(* IEC 61131-3 sources: JaccoSigma/tempclass/Class/VST011 (part 2) *)

      //LowLomit
      if FrequencyLimit8 > FrequencyBandwidth / 2 then
        a_FrequencyLimit[3].LimitLow := FrequencyLimit8 - (FrequencyBandwidth / 2);
      else
        a_FrequencyLimit[3].LimitLow := FrequencyLimit8;
      end_if;

      //High Limit
      if FrequencyLimit8 + (FrequencyBandwidth / 2) < 1000000 then
        a_FrequencyLimit[3].LimitHigh  := FrequencyLimit8 + (FrequencyBandwidth / 2);
      else
        a_FrequencyLimit[3].LimitHigh := FrequencyLimit8;
      end_if;

    else

      //Set inactive
      a_FrequencyLimit[3].LimitHigh := a_FrequencyLimit[3].LimitLow := 16#FFFF_FFFF;

    end_if;

  end_if;

  result := input;

END_FUNCTION

FUNCTION VIRTUAL GLOBAL VST011::FrequencyLimit16::Write
  VAR_INPUT
    input (EAX)   : UDINT;
  END_VAR
  VAR_OUTPUT
    result (EAX)  : UDINT;
  END_VAR

  // Max Frequency is 1 Mhz
  IF input > 1000000 & input <> 16#FFFF_FFFF THEN
    input := 1000000;
  END_IF;

  if FrequencyLimit16 <> input then //do we have a new value?

    //Save Input
    FrequencyLimit16 := input;

    //Set new Limit
    WriteParameter(us_ParameterNr:= VST_ASYNC_FREQUENCYLIMIT16, ud_Value:=FrequencyLimit16);

    //Calculate Limits for Hysterese
    //*****************************************************************************
    if FrequencyLimit16 <> 16#FFFF_FFFF then

      //LowLomit
      if FrequencyLimit16 > FrequencyBandwidth / 2 then
        a_FrequencyLimit[4].LimitLow := FrequencyLimit16 - (FrequencyBandwidth / 2);
      else
        a_FrequencyLimit[4].LimitLow := FrequencyLimit16;
      end_if;

      //High Limit
      if FrequencyLimit16 + (FrequencyBandwidth / 2) < 1000000 then
        a_FrequencyLimit[4].LimitHigh  := FrequencyLimit16 + (FrequencyBandwidth / 2);
      else
        a_FrequencyLimit[4].LimitHigh := FrequencyLimit16;
      end_if;

    else

      //Set inactive
      a_FrequencyLimit[4].LimitHigh := a_FrequencyLimit[4].LimitLow := 16#FFFF_FFFF;

    end_if;

  end_if;

  result := input;

END_FUNCTION

FUNCTION VIRTUAL GLOBAL VST011::FrequencyLimit32::Write
  VAR_INPUT
    input (EAX)   : UDINT;
  END_VAR
  VAR_OUTPUT
    result (EAX)  : UDINT;
  END_VAR

  // Max Frequency is 1 Mhz
  IF input > 1000000 & input <> 16#FFFF_FFFF THEN
    input := 1000000;
  END_IF;

  if FrequencyLimit32 <> input then //do we have a new value?

    //Save Input
    FrequencyLimit32 := input;

    //Set new Limit
    WriteParameter(us_ParameterNr:= VST_ASYNC_FREQUENCYLIMIT32, ud_Value:=FrequencyLimit32);

    //Calculate Limits for Hysterese
    //*****************************************************************************
    if FrequencyLimit32 <> 16#FFFF_FFFF then

      //LowLomit
      if FrequencyLimit32 > FrequencyBandwidth / 2 then
        a_FrequencyLimit[5].LimitLow := FrequencyLimit32 - (FrequencyBandwidth / 2);
      else
        a_FrequencyLimit[5].LimitLow := FrequencyLimit32;
      end_if;

      //High Limit
      if FrequencyLimit32 + (FrequencyBandwidth / 2) < 1000000 then
        a_FrequencyLimit[5].LimitHigh  := FrequencyLimit32 + (FrequencyBandwidth / 2);
      else
        a_FrequencyLimit[5].LimitHigh := FrequencyLimit32;
      end_if;

    else

      //Set inactive
      a_FrequencyLimit[5].LimitHigh := a_FrequencyLimit[5].LimitLow := 16#FFFF_FFFF;

    end_if;

  end_if;

  result := input;

END_FUNCTION

FUNCTION VIRTUAL GLOBAL VST011::HWRampdownDeltaFrequency::Write
  VAR_INPUT
    input (EAX)   : DINT;
  END_VAR
  VAR_OUTPUT
    result (EAX)  : DINT;
  END_VAR

  WriteParameter(us_ParameterNr := VST_ASYNC_EXTERNALLOCKDELTAFREQUENCY, ud_Value := input$UDINT);
  result := input;

END_FUNCTION

FUNCTION VIRTUAL GLOBAL VST011::HWRampdownDeltaTime::Write
  VAR_INPUT
    input (EAX)   : DINT;
  END_VAR
  VAR_OUTPUT
    result (EAX)  : DINT;
  END_VAR

  WriteParameter(us_ParameterNr := VST_ASYNC_EXTERNALLOCKDELTATIME, ud_Value := input$UDINT);
  result := input;

END_FUNCTION

FUNCTION GLOBAL VST011::RequestParameter
  VAR_INPUT
    us_ParameterNr  : USINT;
  END_VAR
  VAR_OUTPUT
    retcode   : DINT;
  END_VAR
  VAR
    tmpCounter : USINT;
  END_VAR

  retcode := VST_ERROR_ASYNC_NOERROR;

  if us_ParameterNr <= VST011_MAXASYNCPARAMETER &  us_ReadNumber <= VST011_MAXASYNCPARAMETER then

    // Check if Element is already active
    //*****************************************************************************
    if us_ReadNumber then

      //No Overflow of Buffer (to be Thread-Safe)
      //---------------------------------------------------------------------------
      if us_ReadPosition + us_ReadNumber - 1 <= VST011_MAXASYNCPARAMETER then

        for tmpCounter := us_ReadPosition to us_ReadPosition + us_ReadNumber - 1 do
          if a_ParameterReadRequest[tmpCounter] = us_ParameterNr then
            retcode := VST_ERROR_ASYNC_ALREADYACTIVE;
            return;
          end_if;
        end_for;

      //Overflow of Buffer (to be Thread-Safe)
      //---------------------------------------------------------------------------
      else

        //Check actual Position to End of Buffer
        for tmpCounter := us_ReadPosition to VST011_MAXASYNCPARAMETER do
          if a_ParameterReadRequest[tmpCounter] = us_ParameterNr then
            retcode := VST_ERROR_ASYNC_ALREADYACTIVE;
            return;
          end_if;
        end_for;

        //Check from Zero to actual Element
        for tmpCounter := 0 to us_ReadNumber - VST011_MAXASYNCPARAMETER + us_ReadPosition - 2 do
          if a_ParameterReadRequest[tmpCounter] = us_ParameterNr then
            retcode := VST_ERROR_ASYNC_ALREADYACTIVE;
            return;
          end_if;
        end_for;
      end_if;

    end_if;

    // Save into Queue for asynchronous ReadAccess
    //*****************************************************************************
    if us_ReadPosition + us_ReadNumber <= VST011_MAXASYNCPARAMETER  then
      a_ParameterReadRequest[us_ReadPosition + us_ReadNumber]   := us_ParameterNr;
    else
      a_ParameterReadRequest[us_ReadPosition + us_ReadNumber - VST011_MAXASYNCPARAMETER - 1] := us_ParameterNr;
    end_if;

    us_ReadNumber += 1;
    a_ReadDataBuffer[us_ParameterNr].b_Valid := false;

  else
    retcode := VST_ERROR_ASYNC_INVALIDPARAMETER;
  end_if;

END_FUNCTION

FUNCTION GLOBAL VST011::WriteParameter
  VAR_INPUT
    us_ParameterNr  : USINT;
    ud_Value  : UDINT;
  END_VAR
  VAR_OUTPUT
    retcode   : DINT;
  END_VAR
  VAR
    tmpCounter : USINT;
    pAsyWrData  : ^t_AsyncWriteData;
    pLastWritten: ^t_LastWrittenValues;
    ForEnd : USINT;
  END_VAR

  retcode := VST_ERROR_ASYNC_NOERROR;

  IF (us_ParameterNr <= VST011_MAXASYNCPARAMETER) & (us_WriteNumber <= VST011_MAXASYNCPARAMETER) THEN
    CASE us_ParameterNr OF
      VST_ASYNC_INCREMENTALENCODERSETTINGS, //not implemented (user otherwise might access internal test-registers)
      VST_ASYNC_BRIDGE2OFF, //implemented but may not be called (user could damage the card)!
      VST_ASYNC_BRIDGE2MUL,
      VST_ASYNC_BRIDGE2DIV,
      VST_ASYNC_BRIDGE1OFF,
      VST_ASYNC_BRIDGE1MUL,
      VST_ASYNC_BRIDGE1DIV,
      VST_ASYNC_BRIDGESUPPLYVOLTAGELOWERTHRESHOLD,
      VST_ASYNC_BRIDGESUPPLYVOLTAGEUPPERTHRESHOLD,
      VST_ASYNC_BRIDGETEMPERATUREWARNINGTHRESHOLD,
      VST_ASYNC_BRIDGETEMPERATUREERRORTHRESHOLD,
      VST_ASYNC_EXTENDEDSTATEWORD,
      VST_ASYNC_COMMUTATIONCOUNTERBRIDGE1,
      VST_ASYNC_COMMUTATIONCOUNTERBRIDGE2,
      VST_ASYNC_ONTIMECOUNTERBRIDGE1,
      VST_ASYNC_ONTIMECOUNTERBRIDGE2,
      VST_ASYNC_HBRIDGE_VOLTAGE,
      VST_ASYNC_HBRIDGE_TEMPERATURE:
        retcode := VST_ERROR_ASYNC_WRITENOTALLOWED;
    ELSE
      // if the value is the same as the last value we wrote on this parameter => don't do it
      pLastWritten := #a_LastWrittenAsyValues[0] + us_ParameterNr * sizeof(t_LastWrittenValues);
      if (pLastWritten^.AlreadyUsed = TRUE) & (ud_Value = pLastWritten^.Value) then
        // this is already the actual value of this parameter
        return;
      end_if;

      // Check if Element is already active
      //*****************************************************************************
      if us_WriteNumber then

        //No Overflow of Buffer (to be Thread-Safe)
        //---------------------------------------------------------------------------
        if us_WritePosition + us_WriteNumber - 1 <= VST011_MAXASYNCPARAMETER then
          // calculate the end only once
          ForEnd := (us_WritePosition + us_WriteNumber - 1);
          pAsyWrData := #a_WriteDataBuffer[0] + us_WritePosition * sizeof(t_AsyncWriteData);
          for tmpCounter := us_WritePosition to ForEnd do
            if pAsyWrData^.us_ID = us_ParameterNr then
              retcode := VST_ERROR_ASYNC_ALREADYACTIVE;
              pAsyWrData^.ud_Value := ud_Value;
              return;
            end_if;
            pAsyWrData += sizeof(a_WriteDataBuffer);
          end_for;

        //Overflow of Buffer (to be Thread-Safe)
        //---------------------------------------------------------------------------
        else
          //Check actual Position to End of Buffer
          pAsyWrData := #a_WriteDataBuffer[0] + us_WritePosition * sizeof(t_AsyncWriteData);
          for tmpCounter := us_WritePosition to VST011_MAXASYNCPARAMETER do
            if pAsyWrData^.us_ID = us_ParameterNr then
              retcode := VST_ERROR_ASYNC_ALREADYACTIVE;
              pAsyWrData^.ud_Value := ud_Value;
              return;
            end_if;
            pAsyWrData += sizeof(t_AsyncWriteData);
          end_for;

          //Check from Zero to actual Element
          ForEnd := us_WriteNumber - VST011_MAXASYNCPARAMETER + us_WritePosition - 2;
          pAsyWrData := #a_WriteDataBuffer[0];
          for tmpCounter := 0 to ForEnd do
            if pAsyWrData^.us_ID = us_ParameterNr then
              retcode := VST_ERROR_ASYNC_ALREADYACTIVE;
              pAsyWrData^.ud_Value := ud_Value;
              return;
            end_if;
            pAsyWrData += sizeof(t_AsyncWriteData);
          end_for;
        end_if;

      end_if;

      // Save into Queue for asynchronous WriteAccess
      //*****************************************************************************
      if us_WritePosition + us_WriteNumber <= VST011_MAXASYNCPARAMETER  then
        pAsyWrData := #a_WriteDataBuffer[0] + (us_WritePosition + us_WriteNumber) * sizeof(t_AsyncWriteData);
      else
        pAsyWrData := #a_WriteDataBuffer[0] + (us_WriteNumber + us_WritePosition - VST011_MAXASYNCPARAMETER - 1) * sizeof(t_AsyncWriteData);
      end_if;

      pAsyWrData^.us_ID    := us_ParameterNr;
      pAsyWrData^.ud_Value := ud_Value;

      pLastWritten^.Value := ud_Value;
      pLastWritten^.AlreadyUsed := TRUE;

      us_WriteNumber += 1;
    END_CASE;
  ELSE
    retcode := VST_ERROR_ASYNC_INVALIDPARAMETER;
  END_IF;

END_FUNCTION

FUNCTION GLOBAL VST011::ReadParameter
  VAR_INPUT
    us_ParameterNr  : USINT;
    p_b_Valid   : ^BOOL;
    p_ud_Value  : ^UDINT;
  END_VAR
  VAR_OUTPUT
    retcode   : DINT;
  END_VAR

  retcode := VST_ERROR_ASYNC_NOERROR;

  IF us_ParameterNr <= VST011_MAXASYNCPARAMETER THEN
    IF p_b_Valid <> NIL THEN
      p_b_Valid^ := a_ReadDataBuffer[us_ParameterNr].b_Valid;
    END_IF;
    a_ReadDataBuffer[us_ParameterNr].b_Valid := FALSE;
    IF p_ud_Value <> NIL THEN
      p_ud_Value^ := a_ReadDataBuffer[us_ParameterNr].ud_Value;
    ELSE
      retcode := VST_ERROR_ASYNC_NOVALUEPTR;
    END_IF;
  ELSE
    retcode := VST_ERROR_ASYNC_INVALIDPARAMETER;
  END_IF;

END_FUNCTION

FUNCTION VIRTUAL GLOBAL VST011::MaxCurrent::Write
  VAR_INPUT
    input (EAX)   : DINT;
  END_VAR
  VAR_OUTPUT
    result (EAX)  : DINT;
  END_VAR

  //Check for Change
  if input <> MaxCurrent then

    //Check Limit
    if input < 0 then
      input := 0;
    elsif input > sd_MaxAllowedCurrent then
      input := sd_MaxAllowedCurrent;
    end_if;

    //Calculate Current
    if abs(SetFreqOut)$UDINT <= udStallCurrentWindow then
      u_MaxCurrent := to_uint(input - ((input * StallCurrentReduction) / 1000));
    else
      u_MaxCurrent := to_uint(input);
    end_if;

  end_if;

  result := MaxCurrent := input;

END_FUNCTION

FUNCTION VIRTUAL GLOBAL VST011::UpdateRetryCounter
  VAR
    tempRetryCounter : USINT;
  END_VAR

  // LanSte 16.04.2013 10:49
  // Updated to use new Method for Payload support
  tempRetryCounter := GetRetryCounter(ud_DOHandle := s_IODataObject.p_Handle$UDINT);
  if ( tempRetryCounter <> s_IODataObject.us_OldRetryCounter ) then
    RetryCounter += TO_USINT( tempRetryCounter - s_IODataObject.us_OldRetryCounter );
    s_IODataObject.us_OldRetryCounter := tempRetryCounter;
  end_if;

  tempRetryCounter := GetRetryCounter(ud_DOHandle := s_ISyncDO.p_Handle$UDINT);
  if ( tempRetryCounter <> s_ISyncDO.us_OldRetryCounter ) then
    RetryCounter += TO_USINT( tempRetryCounter - s_ISyncDO.us_OldRetryCounter );
    s_ISyncDO.us_OldRetryCounter := tempRetryCounter;
  end_if;

  tempRetryCounter := GetRetryCounter(ud_DOHandle := s_SettingsDataObject.p_Handle$UDINT);
  if ( tempRetryCounter <> s_SettingsDataObject.us_OldRetryCounter ) then
    RetryCounter += TO_USINT( tempRetryCounter - s_SettingsDataObject.us_OldRetryCounter );
    s_SettingsDataObject.us_OldRetryCounter := tempRetryCounter;
  end_if;

END_FUNCTION

FUNCTION VIRTUAL GLOBAL VST011::Input1LatchedRising::Read
  VAR_OUTPUT
    output (EAX)  : DINT;
  END_VAR

  output := Input1LatchedRising;
  Input1LatchedRising := 0;

END_FUNCTION

FUNCTION VIRTUAL GLOBAL VST011::Input1LatchedFalling::Read
  VAR_OUTPUT
    output (EAX)  : DINT;
  END_VAR

  output := Input1LatchedFalling;
  Input1LatchedFalling := 0;

END_FUNCTION

FUNCTION VIRTUAL GLOBAL VST011::Input2LatchedRising::Read
  VAR_OUTPUT
    output (EAX)  : DINT;
  END_VAR

  output := Input2LatchedRising;
  Input2LatchedRising := 0;

END_FUNCTION

FUNCTION VIRTUAL GLOBAL VST011::Input2LatchedFalling::Read
  VAR_OUTPUT
    output (EAX)  : DINT;
  END_VAR

  output := Input2LatchedFalling;
  Input2LatchedFalling := 0;

END_FUNCTION

FUNCTION VIRTUAL GLOBAL VST011::ZeroPulse_latched::Read
  VAR_OUTPUT
    output (EAX)  : DINT;
  END_VAR

  output := ZeroPulse_latched;
  ZeroPulse_latched := 0;

END_FUNCTION

FUNCTION VIRTUAL GLOBAL VST011::HWEnableSoftwareRampdown::Write
  VAR_INPUT
    input (EAX)   : DINT;
  END_VAR
  VAR_OUTPUT
    result (EAX)  : DINT;
  END_VAR

  IF input THEN
    HWEnableSoftwareRampdown := 1;
  ELSE
    HWEnableSoftwareRampdown := 0;
  END_IF;
  result := HWEnableSoftwareRampdown;

END_FUNCTION

FUNCTION VIRTUAL GLOBAL VST011::FrequencyBandwidth::Write
  VAR_INPUT
    input (EAX)   : UDINT;
  END_VAR
  VAR_OUTPUT
    result (EAX)  : UDINT;
  END_VAR

  if FrequencyBandwidth <> input then //just do something, if the values differ

    FrequencyBandwidth := input;

    //Calculate FrequencyLimits for Hysterese
    CalcFrequencyLimits();

  end_if;

  result := FrequencyBandwidth;

END_FUNCTION

FUNCTION VIRTUAL GLOBAL VST011::StallCurrentReduction::Write
  VAR_INPUT
    input (EAX)   : DINT;
  END_VAR
  VAR_OUTPUT
    result (EAX)  : DINT;
  END_VAR

  if input <> StallCurrentReduction then //just do something when the value changes

    StallCurrentReduction := input;

    //Check for Limits
    if StallCurrentReduction < 0 then
      StallCurrentReduction := 0;
    elsif StallCurrentReduction > 1000 then
      StallCurrentReduction := 1000;
    end_if;

    //Calculate Current
    if abs(SetFreqOut)$UDINT <= udStallCurrentWindow then
      u_MaxCurrent := to_uint(MaxCurrent - ((MaxCurrent * StallCurrentReduction) / 1000));
    else
      u_MaxCurrent := to_uint(MaxCurrent);
    end_if;

  end_if;

  result := StallCurrentReduction;

END_FUNCTION

FUNCTION VST011::WriteAsyncParameter

  // check if any asynchronous Parameter must be sent
  //*****************************************************************************
  if us_WriteNumber then

    //*****************************************************************************
    //** Depending of the ParameterID, access another Register                   **
    //*****************************************************************************
    case a_WriteDataBuffer[us_WritePosition].us_ID of

     //*****************************************************************************

      VST_ASYNC_CHOPPEROFFTIME:
        s_SettingsDataObject.p_DataWrite$^UINT^ := a_WriteDataBuffer[us_WritePosition].ud_Value$UINT;
        ChopperOffTime$UINT := a_WriteDataBuffer[us_WritePosition].ud_Value$UINT;
        a_ReadDataBuffer[VST_ASYNC_CHOPPEROFFTIME].b_Valid := false;

        AsyWriteAddress(udAddress := VST011_OFFSET_SETTINGS + t_s_SettingsDataType.ChopperOffTime,
                        usLength  := sizeof(t_s_SettingsDataType.ChopperOffTime));

      //*****************************************************************************

      VST_ASYNC_FASTDECAYTIME:
        s_SettingsDataObject.p_DataWrite$^UINT^ := a_WriteDataBuffer[us_WritePosition].ud_Value$UINT;
        FastDecayTime$UINT := a_WriteDataBuffer[us_WritePosition].ud_Value$UINT;
        a_ReadDataBuffer[VST_ASYNC_FASTDECAYTIME].b_Valid := false;

        AsyWriteAddress(udAddress := VST011_OFFSET_SETTINGS + t_s_SettingsDataType.FastDecayTime,
                        usLength  := sizeof(t_s_SettingsDataType.FastDecayTime));

      //*****************************************************************************

      VST_ASYNC_FREQUENCYLIMIT32:
        s_SettingsDataObject.p_DataWrite$^UDINT^ := a_WriteDataBuffer[us_WritePosition].ud_Value;

        if FrequencyBandwidth = 0 then
          FrequencyLimit32 := a_WriteDataBuffer[us_WritePosition].ud_Value;
        end_if;

        a_ReadDataBuffer[VST_ASYNC_FREQUENCYLIMIT32].b_Valid := false;

        AsyWriteAddress(udAddress := VST011_OFFSET_SETTINGS + t_s_SettingsDataType.FrequencyLimit32,
                        usLength  := sizeof(t_s_SettingsDataType.FrequencyLimit32));

      //*****************************************************************************

      VST_ASYNC_FREQUENCYLIMIT16:
        s_SettingsDataObject.p_DataWrite$^UDINT^ := a_WriteDataBuffer[us_WritePosition].ud_Value;

        if FrequencyBandwidth = 0 then
          FrequencyLimit16 := a_WriteDataBuffer[us_WritePosition].ud_Value;
        end_if;

        a_ReadDataBuffer[VST_ASYNC_FREQUENCYLIMIT16].b_Valid := false;

        AsyWriteAddress(udAddress := VST011_OFFSET_SETTINGS + t_s_SettingsDataType.FrequencyLimit16,
                        usLength  := sizeof(t_s_SettingsDataType.FrequencyLimit16));

      //*****************************************************************************

      VST_ASYNC_FREQUENCYLIMIT8:
        s_SettingsDataObject.p_DataWrite$^UDINT^ := a_WriteDataBuffer[us_WritePosition].ud_Value;

        if FrequencyBandwidth = 0 then
          FrequencyLimit8 := a_WriteDataBuffer[us_WritePosition].ud_Value;
        end_if;

        a_ReadDataBuffer[VST_ASYNC_FREQUENCYLIMIT8].b_Valid := false;

        AsyWriteAddress(udAddress := VST011_OFFSET_SETTINGS + t_s_SettingsDataType.FrequencyLimit8,
                        usLength  := sizeof(t_s_SettingsDataType.FrequencyLimit8));

      //*****************************************************************************

      VST_ASYNC_FREQUENCYLIMIT4:
        s_SettingsDataObject.p_DataWrite$^UDINT^ := a_WriteDataBuffer[us_WritePosition].ud_Value;

        if FrequencyBandwidth = 0 then
          FrequencyLimit4 := a_WriteDataBuffer[us_WritePosition].ud_Value;
        end_if;

        a_ReadDataBuffer[VST_ASYNC_FREQUENCYLIMIT4].b_Valid := false;

        AsyWriteAddress(udAddress := VST011_OFFSET_SETTINGS + t_s_SettingsDataType.FrequencyLimit4,
                        usLength  := sizeof(t_s_SettingsDataType.FrequencyLimit4));

      //*****************************************************************************

      VST_ASYNC_FREQUENCYLIMIT2:
        s_SettingsDataObject.p_DataWrite$^UDINT^ := a_WriteDataBuffer[us_WritePosition].ud_Value;

        if FrequencyBandwidth = 0 then
          FrequencyLimit2:= a_WriteDataBuffer[us_WritePosition].ud_Value;
        end_if;

        a_ReadDataBuffer[VST_ASYNC_FREQUENCYLIMIT2].b_Valid := false;

        AsyWriteAddress(udAddress := VST011_OFFSET_SETTINGS + t_s_SettingsDataType.FrequencyLimit2,
                        usLength  := sizeof(t_s_SettingsDataType.FrequencyLimit2));

      //*****************************************************************************

      VST_ASYNC_FREQUENCYLIMIT1:
        s_SettingsDataObject.p_DataWrite$^UDINT^ := a_WriteDataBuffer[us_WritePosition].ud_Value;

        if FrequencyBandwidth = 0 then
          FrequencyLimit1:= a_WriteDataBuffer[us_WritePosition].ud_Value;
        end_if;

        a_ReadDataBuffer[VST_ASYNC_FREQUENCYLIMIT1].b_Valid := false;

        AsyWriteAddress(udAddress := VST011_OFFSET_SETTINGS + t_s_SettingsDataType.FrequencyLimit1,
                        usLength  := sizeof(t_s_SettingsDataType.FrequencyLimit1));

      //*****************************************************************************

      VST_ASYNC_EXTERNALLOCKDELTAFREQUENCY:
        s_SettingsDataObject.p_DataWrite$^UINT^ := a_WriteDataBuffer[us_WritePosition].ud_Value$UINT;
        HWRampdownDeltaFrequency$UINT := a_WriteDataBuffer[us_WritePosition].ud_Value$UINT;
        a_ReadDataBuffer[VST_ASYNC_EXTERNALLOCKDELTAFREQUENCY].b_Valid := false;

        AsyWriteAddress(udAddress := VST011_OFFSET_SETTINGS + t_s_SettingsDataType.HWRampdownDeltaFrequency,
                        usLength  := sizeof(t_s_SettingsDataType.HWRampdownDeltaFrequency));

      //*****************************************************************************

      VST_ASYNC_EXTERNALLOCKDELTATIME:
        s_SettingsDataObject.p_DataWrite$^UINT^ := a_WriteDataBuffer[us_WritePosition].ud_Value$UINT;
        HWRampdownDeltaTime$UINT := a_WriteDataBuffer[us_WritePosition].ud_Value$UINT;
        a_ReadDataBuffer[VST_ASYNC_EXTERNALLOCKDELTATIME].b_Valid := false;

        AsyWriteAddress(udAddress := VST011_OFFSET_SETTINGS + t_s_SettingsDataType.HWRampdownDeltaTime,
                        usLength  := sizeof(t_s_SettingsDataType.HWRampdownDeltaTime));

      //*****************************************************************************

      VST_ASYNC_INCREMENTALENCODERSETTINGS:
        //** not implemented    *******************************************************

      //*****************************************************************************

      VST_ASYNC_BLANKINGTIMEREGISTER:
        s_SettingsDataObject.p_DataWrite$^UINT^ := a_WriteDataBuffer[us_WritePosition].ud_Value$UINT;
        BlankingTime$UINT := a_WriteDataBuffer[us_WritePosition].ud_Value$UINT;
        a_ReadDataBuffer[VST_ASYNC_BLANKINGTIMEREGISTER].b_Valid := false;

        AsyWriteAddress(udAddress := VST011_OFFSET_SETTINGS + t_s_SettingsDataType.BlankingTimeRegister,
                        usLength  := sizeof(t_s_SettingsDataType.BlankingTimeRegister));

      //*****************************************************************************

      VST_ASYNC_BRIDGE2OFF:
        s_SettingsDataObject.p_DataWrite$^UINT^ := a_WriteDataBuffer[us_WritePosition].ud_Value$UINT;
        a_ReadDataBuffer[VST_ASYNC_BRIDGE2OFF].b_Valid := false;

        AsyWriteAddress(udAddress := VST011_OFFSET_SETTINGS + t_s_SettingsDataType.Bridge2Off,
                        usLength  := sizeof(t_s_SettingsDataType.Bridge2Off));

      //*****************************************************************************

      VST_ASYNC_BRIDGE2MUL:
        s_SettingsDataObject.p_DataWrite$^UINT^ := a_WriteDataBuffer[us_WritePosition].ud_Value$UINT;
        a_ReadDataBuffer[VST_ASYNC_BRIDGE2MUL].b_Valid := false;

        AsyWriteAddress(udAddress := VST011_OFFSET_SETTINGS + t_s_SettingsDataType.Bridge2Mul,
                        usLength  := sizeof(t_s_SettingsDataType.Bridge2Mul));

      //*****************************************************************************

      VST_ASYNC_BRIDGE2DIV:
        s_SettingsDataObject.p_DataWrite$^UINT^ := a_WriteDataBuffer[us_WritePosition].ud_Value$UINT;
        a_ReadDataBuffer[VST_ASYNC_BRIDGE2DIV].b_Valid := false;

        AsyWriteAddress(udAddress := VST011_OFFSET_SETTINGS + t_s_SettingsDataType.Bridge2Div,
                        usLength  := sizeof(t_s_SettingsDataType.Bridge2Div));

      //*****************************************************************************

      VST_ASYNC_BRIDGE1OFF:
        s_SettingsDataObject.p_DataWrite$^UINT^ := a_WriteDataBuffer[us_WritePosition].ud_Value$UINT;
        a_ReadDataBuffer[VST_ASYNC_BRIDGE1OFF].b_Valid := false;

        AsyWriteAddress(udAddress := VST011_OFFSET_SETTINGS + t_s_SettingsDataType.Bridge1Off,
                        usLength  := sizeof(t_s_SettingsDataType.Bridge1Off));

      //*****************************************************************************

      VST_ASYNC_BRIDGE1MUL:
        s_SettingsDataObject.p_DataWrite$^UINT^ := a_WriteDataBuffer[us_WritePosition].ud_Value$UINT;
        a_ReadDataBuffer[VST_ASYNC_BRIDGE1MUL].b_Valid := false;

        AsyWriteAddress(udAddress := VST011_OFFSET_SETTINGS + t_s_SettingsDataType.Bridge1Mul,
                        usLength  := sizeof(t_s_SettingsDataType.Bridge1Mul));

      //*****************************************************************************

      VST_ASYNC_BRIDGE1DIV:
        s_SettingsDataObject.p_DataWrite$^UINT^ := a_WriteDataBuffer[us_WritePosition].ud_Value$UINT;
        a_ReadDataBuffer[VST_ASYNC_BRIDGE1DIV].b_Valid := false;

        AsyWriteAddress(udAddress := VST011_OFFSET_SETTINGS + t_s_SettingsDataType.Bridge1Div,
                        usLength  := sizeof(t_s_SettingsDataType.Bridge1Div));

      //*****************************************************************************

      VST_ASYNC_BRIDGESUPPLYVOLTAGELOWERTHRESHOLD:
        s_SettingsDataObject.p_DataWrite$^UINT^ := a_WriteDataBuffer[us_WritePosition].ud_Value$UINT;
        a_ReadDataBuffer[VST_ASYNC_BRIDGESUPPLYVOLTAGELOWERTHRESHOLD].b_Valid := false;

        AsyWriteAddress(udAddress := VST011_OFFSET_SETTINGS + t_s_SettingsDataType.BridgeSupplyVoltageLowerThreshold,
                        usLength  := sizeof(t_s_SettingsDataType.BridgeSupplyVoltageLowerThreshold));

      //*****************************************************************************

      VST_ASYNC_BRIDGESUPPLYVOLTAGEUPPERTHRESHOLD:
        s_SettingsDataObject.p_DataWrite$^UINT^ := a_WriteDataBuffer[us_WritePosition].ud_Value$UINT;
        a_ReadDataBuffer[VST_ASYNC_BRIDGESUPPLYVOLTAGEUPPERTHRESHOLD].b_Valid := false;

        AsyWriteAddress(udAddress := VST011_OFFSET_SETTINGS + t_s_SettingsDataType.BridgeSupplyVoltageUpperThreshold,
                        usLength  := sizeof(t_s_SettingsDataType.BridgeSupplyVoltageUpperThreshold));

      //*****************************************************************************

      VST_ASYNC_BRIDGETEMPERATUREWARNINGTHRESHOLD:
        s_SettingsDataObject.p_DataWrite$^UINT^ := a_WriteDataBuffer[us_WritePosition].ud_Value$UINT;
        a_ReadDataBuffer[VST_ASYNC_BRIDGETEMPERATUREWARNINGTHRESHOLD].b_Valid := false;

        AsyWriteAddress(udAddress := VST011_OFFSET_SETTINGS + t_s_SettingsDataType.BridgeTemperatureWarningThreshold,
                        usLength  := sizeof(t_s_SettingsDataType.BridgeTemperatureWarningThreshold));

      //*****************************************************************************

      VST_ASYNC_BRIDGETEMPERATUREERRORTHRESHOLD:
        s_SettingsDataObject.p_DataWrite$^UINT^ := a_WriteDataBuffer[us_WritePosition].ud_Value$UINT;
        a_ReadDataBuffer[VST_ASYNC_BRIDGETEMPERATUREERRORTHRESHOLD].b_Valid := false;

        AsyWriteAddress(udAddress := VST011_OFFSET_SETTINGS + t_s_SettingsDataType.BridgeTemperatureErrorThreshold,
                        usLength  := sizeof(t_s_SettingsDataType.BridgeTemperatureErrorThreshold));

      //*****************************************************************************

    end_case;

    // One Element is done
    us_WritePosition  += 1;

    // Handle Overflow of Bufferposition
    if us_WritePosition > VST011_MAXASYNCPARAMETER then
      us_WritePosition := 0;
    end_if;

    us_WriteNumber    -= 1;
  end_if;

END_FUNCTION

FUNCTION VST011::ReadAsyncParameter
VAR
  tmpValue : DINT;
END_VAR

  //*****************************************************************************
  //** check if we requested data in last cycle                                **
  //*****************************************************************************
  if us_ParameterReadRequestActive then

    case us_ParameterReadRequestActive - 1 of

      //*****************************************************************************

      VST_ASYNC_CHOPPEROFFTIME:
        a_ReadDataBuffer[VST_ASYNC_CHOPPEROFFTIME].ud_Value := to_UDINT(s_SettingsDataObject.p_DataRead$^UINT^);
        a_ReadDataBuffer[VST_ASYNC_CHOPPEROFFTIME].b_Valid := TRUE;

      //*****************************************************************************

      VST_ASYNC_FASTDECAYTIME:
        a_ReadDataBuffer[VST_ASYNC_FASTDECAYTIME].ud_Value := to_UDINT(s_SettingsDataObject.p_DataRead$^UINT^);
        a_ReadDataBuffer[VST_ASYNC_FASTDECAYTIME].b_Valid := TRUE;

      //*****************************************************************************

      VST_ASYNC_FREQUENCYLIMIT32:
        a_ReadDataBuffer[VST_ASYNC_FREQUENCYLIMIT32].ud_Value := s_SettingsDataObject.p_DataRead^;
        a_ReadDataBuffer[VST_ASYNC_FREQUENCYLIMIT32].b_Valid := TRUE;

      //*****************************************************************************

      VST_ASYNC_FREQUENCYLIMIT16:
        a_ReadDataBuffer[VST_ASYNC_FREQUENCYLIMIT16].ud_Value := s_SettingsDataObject.p_DataRead^;
        a_ReadDataBuffer[VST_ASYNC_FREQUENCYLIMIT16].b_Valid := TRUE;

      //*****************************************************************************

      VST_ASYNC_FREQUENCYLIMIT8:
        a_ReadDataBuffer[VST_ASYNC_FREQUENCYLIMIT8].ud_Value := s_SettingsDataObject.p_DataRead^;
        a_ReadDataBuffer[VST_ASYNC_FREQUENCYLIMIT8].b_Valid := TRUE;

      //*****************************************************************************

      VST_ASYNC_FREQUENCYLIMIT4:
        a_ReadDataBuffer[VST_ASYNC_FREQUENCYLIMIT4].ud_Value := s_SettingsDataObject.p_DataRead^;
        a_ReadDataBuffer[VST_ASYNC_FREQUENCYLIMIT4].b_Valid := TRUE;

      //*****************************************************************************

      VST_ASYNC_FREQUENCYLIMIT2:
        a_ReadDataBuffer[VST_ASYNC_FREQUENCYLIMIT2].ud_Value := s_SettingsDataObject.p_DataRead^;
        a_ReadDataBuffer[VST_ASYNC_FREQUENCYLIMIT2].b_Valid := TRUE;

      //*****************************************************************************

      VST_ASYNC_FREQUENCYLIMIT1:
        a_ReadDataBuffer[VST_ASYNC_FREQUENCYLIMIT1].ud_Value := s_SettingsDataObject.p_DataRead^;
        a_ReadDataBuffer[VST_ASYNC_FREQUENCYLIMIT1].b_Valid := TRUE;

      //*****************************************************************************

      VST_ASYNC_EXTERNALLOCKDELTAFREQUENCY:
        a_ReadDataBuffer[VST_ASYNC_EXTERNALLOCKDELTAFREQUENCY].ud_Value := s_SettingsDataObject.p_DataRead$^UINT^;
        a_ReadDataBuffer[VST_ASYNC_EXTERNALLOCKDELTAFREQUENCY].b_Valid := TRUE;

      //*****************************************************************************

      VST_ASYNC_EXTERNALLOCKDELTATIME:
        a_ReadDataBuffer[VST_ASYNC_EXTERNALLOCKDELTATIME].ud_Value := to_UDINT(s_SettingsDataObject.p_DataRead$^UINT^);
        a_ReadDataBuffer[VST_ASYNC_EXTERNALLOCKDELTATIME].b_Valid := TRUE;

      //*****************************************************************************

      VST_ASYNC_INCREMENTALENCODERSETTINGS:
        a_ReadDataBuffer[VST_ASYNC_INCREMENTALENCODERSETTINGS].ud_Value := to_UDINT(s_SettingsDataObject.p_DataRead$^USINT^);
        a_ReadDataBuffer[VST_ASYNC_INCREMENTALENCODERSETTINGS].b_Valid := TRUE;

      //*****************************************************************************

      VST_ASYNC_BLANKINGTIMEREGISTER:
        a_ReadDataBuffer[VST_ASYNC_BLANKINGTIMEREGISTER].ud_Value := to_UDINT(s_SettingsDataObject.p_DataRead$^USINT^);
        a_ReadDataBuffer[VST_ASYNC_BLANKINGTIMEREGISTER].b_Valid := TRUE;

      //*****************************************************************************

      VST_ASYNC_BRIDGE2OFF:
        a_ReadDataBuffer[VST_ASYNC_BRIDGE2OFF].ud_Value := to_UDINT(s_SettingsDataObject.p_DataRead$^UINT^);
        a_ReadDataBuffer[VST_ASYNC_BRIDGE2OFF].b_Valid := TRUE;

      //*****************************************************************************

      VST_ASYNC_BRIDGE2MUL:
        a_ReadDataBuffer[VST_ASYNC_BRIDGE2MUL].ud_Value := to_UDINT(s_SettingsDataObject.p_DataRead$^UINT^);
        a_ReadDataBuffer[VST_ASYNC_BRIDGE2MUL].b_Valid := TRUE;

      //*****************************************************************************

      VST_ASYNC_BRIDGE2DIV:
        a_ReadDataBuffer[VST_ASYNC_BRIDGE2DIV].ud_Value := to_UDINT(s_SettingsDataObject.p_DataRead$^UINT^);
        a_ReadDataBuffer[VST_ASYNC_BRIDGE2DIV].b_Valid := TRUE;

      //*****************************************************************************

      VST_ASYNC_BRIDGE1OFF:
        a_ReadDataBuffer[VST_ASYNC_BRIDGE1OFF].ud_Value := to_UDINT(s_SettingsDataObject.p_DataRead$^UINT^);
        a_ReadDataBuffer[VST_ASYNC_BRIDGE1OFF].b_Valid := TRUE;

      //*****************************************************************************

      VST_ASYNC_BRIDGE1MUL:
        a_ReadDataBuffer[VST_ASYNC_BRIDGE1MUL].ud_Value := to_UDINT(s_SettingsDataObject.p_DataRead$^UINT^);
        a_ReadDataBuffer[VST_ASYNC_BRIDGE1MUL].b_Valid := TRUE;

      //*****************************************************************************

      VST_ASYNC_BRIDGE1DIV:
        a_ReadDataBuffer[VST_ASYNC_BRIDGE1DIV].ud_Value := to_UDINT(s_SettingsDataObject.p_DataRead$^UINT^);
        a_ReadDataBuffer[VST_ASYNC_BRIDGE1DIV].b_Valid := TRUE;

      //*****************************************************************************

      VST_ASYNC_BRIDGESUPPLYVOLTAGELOWERTHRESHOLD:
        a_ReadDataBuffer[VST_ASYNC_BRIDGESUPPLYVOLTAGELOWERTHRESHOLD].ud_Value := to_UDINT(s_SettingsDataObject.p_DataRead$^UINT^);
        a_ReadDataBuffer[VST_ASYNC_BRIDGESUPPLYVOLTAGELOWERTHRESHOLD].b_Valid := TRUE;

      //*****************************************************************************

      VST_ASYNC_BRIDGESUPPLYVOLTAGEUPPERTHRESHOLD:
        a_ReadDataBuffer[VST_ASYNC_BRIDGESUPPLYVOLTAGEUPPERTHRESHOLD].ud_Value := to_UDINT(s_SettingsDataObject.p_DataRead$^UINT^);
        a_ReadDataBuffer[VST_ASYNC_BRIDGESUPPLYVOLTAGEUPPERTHRESHOLD].b_Valid := TRUE;

      //*****************************************************************************

      VST_ASYNC_BRIDGETEMPERATUREWARNINGTHRESHOLD:
        a_ReadDataBuffer[VST_ASYNC_BRIDGETEMPERATUREWARNINGTHRESHOLD].ud_Value := to_UDINT(s_SettingsDataObject.p_DataRead$^UINT^);
        a_ReadDataBuffer[VST_ASYNC_BRIDGETEMPERATUREWARNINGTHRESHOLD].b_Valid := TRUE;

      //*****************************************************************************

      VST_ASYNC_BRIDGETEMPERATUREERRORTHRESHOLD:
        a_ReadDataBuffer[VST_ASYNC_BRIDGETEMPERATUREERRORTHRESHOLD].ud_Value := to_UDINT(s_SettingsDataObject.p_DataRead$^UINT^);
        a_ReadDataBuffer[VST_ASYNC_BRIDGETEMPERATUREERRORTHRESHOLD].b_Valid := TRUE;

      //*****************************************************************************

      VST_ASYNC_EXTENDEDSTATEWORD:
        a_ReadDataBuffer[VST_ASYNC_EXTENDEDSTATEWORD].ud_Value := to_UDINT(s_SettingsDataObject.p_DataRead$^UINT^);
        a_ReadDataBuffer[VST_ASYNC_EXTENDEDSTATEWORD].b_Valid := TRUE;

      //*****************************************************************************

      VST_ASYNC_COMMUTATIONCOUNTERBRIDGE1:
        a_ReadDataBuffer[VST_ASYNC_COMMUTATIONCOUNTERBRIDGE1].ud_Value := to_UDINT(s_SettingsDataObject.p_DataRead$^UINT^);
        a_ReadDataBuffer[VST_ASYNC_COMMUTATIONCOUNTERBRIDGE1].b_Valid := TRUE;

      //*****************************************************************************

      VST_ASYNC_COMMUTATIONCOUNTERBRIDGE2:
        a_ReadDataBuffer[VST_ASYNC_COMMUTATIONCOUNTERBRIDGE2].ud_Value := to_UDINT(s_SettingsDataObject.p_DataRead$^UINT^);
        a_ReadDataBuffer[VST_ASYNC_COMMUTATIONCOUNTERBRIDGE2].b_Valid := TRUE;

      //*****************************************************************************

      VST_ASYNC_ONTIMECOUNTERBRIDGE1:
        a_ReadDataBuffer[VST_ASYNC_ONTIMECOUNTERBRIDGE1].ud_Value := to_UDINT(s_SettingsDataObject.p_DataRead$^UINT^);
        a_ReadDataBuffer[VST_ASYNC_ONTIMECOUNTERBRIDGE1].b_Valid := TRUE;

      //*****************************************************************************

      VST_ASYNC_ONTIMECOUNTERBRIDGE2:
        a_ReadDataBuffer[VST_ASYNC_ONTIMECOUNTERBRIDGE2].ud_Value := to_UDINT(s_SettingsDataObject.p_DataRead$^UINT^);
        a_ReadDataBuffer[VST_ASYNC_ONTIMECOUNTERBRIDGE2].b_Valid := TRUE;

      //*****************************************************************************

      VST_ASYNC_HBRIDGE_VOLTAGE:
        volt_raw_raw := s_SettingsDataObject.p_DataRead$^HINT^;
        tmpValue := DIV_AB_BY_C(volt_raw_raw + a_CalibData.AI1Offset, a_CalibData.AI1Multiplikator, a_CalibData.AI1Divisor);
        a_ReadDataBuffer[VST_ASYNC_HBRIDGE_VOLTAGE].ud_Value := to_UDINT(tmpValue);
        a_ReadDataBuffer[VST_ASYNC_HBRIDGE_VOLTAGE].b_Valid := TRUE;

      //*****************************************************************************

      VST_ASYNC_HBRIDGE_TEMPERATURE:
        temp_raw_raw := s_SettingsDataObject.p_DataRead$^HINT^;
        tmpValue := DIV_AB_BY_C(temp_raw_raw + a_CalibData.AI2Offset, a_CalibData.AI2Multiplikator, a_CalibData.AI2Divisor);
        a_ReadDataBuffer[VST_ASYNC_HBRIDGE_TEMPERATURE].ud_Value := to_UDINT(tmpValue);
        a_ReadDataBuffer[VST_ASYNC_HBRIDGE_TEMPERATURE].b_Valid := TRUE;

      //*****************************************************************************

    end_case;

    //Request is done
    us_ParameterReadRequestActive := 0;

  end_if;

  // check if any asynchronous Parameter must be read
  //*****************************************************************************
  if us_ReadNumber then

    //*****************************************************************************
    //** Depending of the ParameterID, access another Register                   **
    //*****************************************************************************
    case a_ParameterReadRequest[us_ReadPosition] of

      //*****************************************************************************

      VST_ASYNC_CHOPPEROFFTIME:
        AsyReadAddress( udAddress := VST011_OFFSET_SETTINGS + t_s_SettingsDataType.ChopperOffTime,
                        usLength  := sizeof(t_s_SettingsDataType.ChopperOffTime));

      //*****************************************************************************

      VST_ASYNC_FASTDECAYTIME:
        AsyReadAddress( udAddress := VST011_OFFSET_SETTINGS + t_s_SettingsDataType.FastDecayTime,
                        usLength  := sizeof(t_s_SettingsDataType.FastDecayTime));

      //*****************************************************************************

      VST_ASYNC_FREQUENCYLIMIT32:
        AsyReadAddress( udAddress := VST011_OFFSET_SETTINGS + t_s_SettingsDataType.FrequencyLimit32,
                        usLength  := sizeof(t_s_SettingsDataType.FrequencyLimit32));

      //*****************************************************************************

      VST_ASYNC_FREQUENCYLIMIT16:
        AsyReadAddress( udAddress := VST011_OFFSET_SETTINGS + t_s_SettingsDataType.FrequencyLimit16,
                        usLength  := sizeof(t_s_SettingsDataType.FrequencyLimit16));

      //*****************************************************************************

      VST_ASYNC_FREQUENCYLIMIT8:
        AsyReadAddress( udAddress := VST011_OFFSET_SETTINGS + t_s_SettingsDataType.FrequencyLimit8,
                        usLength  := sizeof(t_s_SettingsDataType.FrequencyLimit8));

      //*****************************************************************************

      VST_ASYNC_FREQUENCYLIMIT4:
        AsyReadAddress( udAddress := VST011_OFFSET_SETTINGS + t_s_SettingsDataType.FrequencyLimit4,
                        usLength  := sizeof(t_s_SettingsDataType.FrequencyLimit4));

      //*****************************************************************************

      VST_ASYNC_FREQUENCYLIMIT2:
        AsyReadAddress( udAddress := VST011_OFFSET_SETTINGS + t_s_SettingsDataType.FrequencyLimit2,
                        usLength  := sizeof(t_s_SettingsDataType.FrequencyLimit2));

      //*****************************************************************************

      VST_ASYNC_FREQUENCYLIMIT1:
        AsyReadAddress(udAddress := VST011_OFFSET_SETTINGS + t_s_SettingsDataType.FrequencyLimit1,
                    usLength  := sizeof(t_s_SettingsDataType.FrequencyLimit1));

      //*****************************************************************************

      VST_ASYNC_EXTERNALLOCKDELTAFREQUENCY:
        AsyReadAddress( udAddress := VST011_OFFSET_SETTINGS + t_s_SettingsDataType.HWRampdownDeltaFrequency,
                        usLength  := sizeof(t_s_SettingsDataType.HWRampdownDeltaFrequency));

      //*****************************************************************************

      VST_ASYNC_EXTERNALLOCKDELTATIME:
        AsyReadAddress( udAddress := VST011_OFFSET_SETTINGS + t_s_SettingsDataType.HWRampdownDeltaTime,
                        usLength  := sizeof(t_s_SettingsDataType.HWRampdownDeltaTime));

      //*****************************************************************************

      VST_ASYNC_INCREMENTALENCODERSETTINGS:
        AsyReadAddress( udAddress := VST011_OFFSET_SETTINGS + t_s_SettingsDataType.IncrementalEncoderSettings,
                        usLength  := sizeof(t_s_SettingsDataType.IncrementalEncoderSettings));

      //*****************************************************************************

      VST_ASYNC_BLANKINGTIMEREGISTER:
        AsyReadAddress( udAddress := VST011_OFFSET_SETTINGS + t_s_SettingsDataType.BlankingTimeRegister,
                        usLength  := sizeof(t_s_SettingsDataType.BlankingTimeRegister));

      //*****************************************************************************

      VST_ASYNC_BRIDGE2OFF:
        AsyReadAddress( udAddress := VST011_OFFSET_SETTINGS + t_s_SettingsDataType.Bridge2Off,
                        usLength  := sizeof(t_s_SettingsDataType.Bridge2Off));

      //*****************************************************************************

      VST_ASYNC_BRIDGE2MUL:
        AsyReadAddress( udAddress := VST011_OFFSET_SETTINGS + t_s_SettingsDataType.Bridge2Mul,
                        usLength  := sizeof(t_s_SettingsDataType.Bridge2Mul));

      //*****************************************************************************

      VST_ASYNC_BRIDGE2DIV:
        AsyReadAddress( udAddress := VST011_OFFSET_SETTINGS + t_s_SettingsDataType.Bridge2Div,
                        usLength  := sizeof(t_s_SettingsDataType.Bridge2Div));

      //*****************************************************************************

      VST_ASYNC_BRIDGE1OFF:
        AsyReadAddress( udAddress := VST011_OFFSET_SETTINGS + t_s_SettingsDataType.Bridge1Off,
                        usLength  := sizeof(t_s_SettingsDataType.Bridge1Off));

      //*****************************************************************************

      VST_ASYNC_BRIDGE1MUL:
        AsyReadAddress( udAddress := VST011_OFFSET_SETTINGS + t_s_SettingsDataType.Bridge1Mul,
                        usLength  := sizeof(t_s_SettingsDataType.Bridge1Mul));

      //*****************************************************************************

      VST_ASYNC_BRIDGE1DIV:
        AsyReadAddress( udAddress := VST011_OFFSET_SETTINGS + t_s_SettingsDataType.Bridge1Div,
                        usLength  := sizeof(t_s_SettingsDataType.Bridge1Div));

      //*****************************************************************************

      VST_ASYNC_BRIDGESUPPLYVOLTAGELOWERTHRESHOLD:
        AsyReadAddress( udAddress := VST011_OFFSET_SETTINGS + t_s_SettingsDataType.BridgeSupplyVoltageLowerThreshold,
                        usLength  := sizeof(t_s_SettingsDataType.BridgeSupplyVoltageLowerThreshold));

      //*****************************************************************************

      VST_ASYNC_BRIDGESUPPLYVOLTAGEUPPERTHRESHOLD:
        AsyReadAddress( udAddress := VST011_OFFSET_SETTINGS + t_s_SettingsDataType.BridgeSupplyVoltageUpperThreshold,
                        usLength  := sizeof(t_s_SettingsDataType.BridgeSupplyVoltageUpperThreshold));

      //*****************************************************************************

      VST_ASYNC_BRIDGETEMPERATUREWARNINGTHRESHOLD:
        AsyReadAddress( udAddress := VST011_OFFSET_SETTINGS + t_s_SettingsDataType.BridgeTemperatureWarningThreshold,
                        usLength  := sizeof(t_s_SettingsDataType.BridgeTemperatureWarningThreshold));

      //*****************************************************************************

      VST_ASYNC_BRIDGETEMPERATUREERRORTHRESHOLD:
        AsyReadAddress( udAddress := VST011_OFFSET_SETTINGS + t_s_SettingsDataType.BridgeTemperatureErrorThreshold,
                        usLength  := sizeof(t_s_SettingsDataType.BridgeTemperatureErrorThreshold));

      //*****************************************************************************

      VST_ASYNC_EXTENDEDSTATEWORD:
        AsyReadAddress( udAddress := 16#50,
                        usLength  := 2);

      //*****************************************************************************

      VST_ASYNC_COMMUTATIONCOUNTERBRIDGE1:
        AsyReadAddress( udAddress := 16#52,
                        usLength  := 2);

      //*****************************************************************************

      VST_ASYNC_COMMUTATIONCOUNTERBRIDGE2:
        AsyReadAddress( udAddress := 16#54,
                        usLength  := 2);

      //*****************************************************************************

      VST_ASYNC_ONTIMECOUNTERBRIDGE1:
        AsyReadAddress( udAddress := 16#56,
                        usLength  := 2);

      //*****************************************************************************

      VST_ASYNC_ONTIMECOUNTERBRIDGE2:
        AsyReadAddress( udAddress := 16#58,
                        usLength  := 2);

      //*****************************************************************************

      VST_ASYNC_HBRIDGE_VOLTAGE:
        AsyReadAddress( udAddress := 16#5A,
                        usLength  := 2);

      //*****************************************************************************

      VST_ASYNC_HBRIDGE_TEMPERATURE:
        AsyReadAddress( udAddress := 16#5C,
                        usLength  := 2);

      //*****************************************************************************

    end_case;

    //Read Request is active
    us_ParameterReadRequestActive := a_ParameterReadRequest[us_ReadPosition] + 1;

    // One Element is done
    us_ReadPosition  += 1;

    // Handle Overflow of Bufferposition
    if us_ReadPosition > VST011_MAXASYNCPARAMETER then
      us_ReadPosition := 0;
    end_if;

    //One Element is done
    us_ReadNumber -= 1;

  end_if;

END_FUNCTION

FUNCTION GLOBAL VST011::ChangeCallMode
  VAR_INPUT
    usID  : USINT;
    bActive   : BOOL;
  END_VAR

  //Check Input-Parameter
  if usID < 0 | usID >= VST_ID_CLASSESAVAILABLE then
    return;
  end_if;

  //Set Call to active
  sAsyCalls[usID].bActive := bActive;

END_FUNCTION

FUNCTION GLOBAL VST011::AddAsyCall
  VAR_INPUT
    usID  : USINT;
    pThis   : ^void;
  END_VAR
  VAR_OUTPUT
    bSuccessful   : BOOL;
  END_VAR

  //Init Returncode
  bSuccessful := false;

  //Check Input-Parameter
  if usID < 0 | usID >= VST_ID_CLASSESAVAILABLE | pThis = NIL then
    return;
  end_if;

  //Already active
  if sAsyCalls[usID].pThis <> NIL then
    return;
  end_if;

  //Add Element
  sAsyCalls[usID].bActive := false;
  sAsyCalls[usID].pThis   := pThis;

  //Everything successful
  bSuccessful := true;

END_FUNCTION

FUNCTION VST011::AsyReadAddress
  VAR_INPUT
    udAddress   : UDINT;
    usLength  : USINT;
  END_VAR

  if b_PayloadSupport then
    // usLengthOfExpAnswer and usSendBufferLength are automatically adjusted to the correct length when us_ByteCntRd and us_ByteCntWr in MULTI_VARAN_i
    ChangeDOLengthOffset( ud_DOHandle           := s_SettingsDataObject.p_Handle$UDINT
                        , ud_offset_read        := udAddress
                        , ud_length_read        := usLength);

    s_SettingsDataObject.b_DOIsRunning.StartRequest := true;
  else
    //Set Address which should be read
    s_SettingsDataObject.p_DOSettings^.ud_AddressRd := DeviceAddress + udAddress;

    //Set Length of Package
    s_SettingsDataObject.p_DOSettings^.us_ByteCntRd := usLength;

    //Set Length of expected Answer
    s_SettingsDataObject.p_Handle^.usLengthofExpAnswer := 1 + usLength;
  end_if;

END_FUNCTION

FUNCTION VST011::AsyWriteAddress
  VAR_INPUT
    udAddress   : UDINT;
    usLength  : USINT;
  END_VAR

  if b_PayloadSupport then
    // usLengthOfExpAnswer and usSendBufferLength are automatically adjusted to the correct length when us_ByteCntRd and us_ByteCntWr in MULTI_VARAN_i
    ChangeDOLengthOffset( ud_DOHandle         := s_SettingsDataObject.p_Handle$UDINT
                        , ud_offset_write     := udAddress
                        , ud_length_write     := usLength);

    s_SettingsDataObject.b_DOIsRunning.StartRequest := true;
  else
    //Set Address which should be written
    s_SettingsDataObject.p_DOSettings^.ud_AddressWr := DeviceAddress + udAddress;

    //Set Length of Package
    s_SettingsDataObject.p_DOSettings^.us_ByteCntWr := usLength;

    //Set Length of Package
    s_SettingsDataObject.p_Handle^.usSendBufferLength :=  11 + usLength;
  end_if;

END_FUNCTION

FUNCTION VST011::IsoReadAddress
  VAR_INPUT
    udAddress   : UDINT;
  END_VAR
  VAR
    s_PropertyValuePair : LSL_PROPERTY_VALUE_PAIR;
  END_VAR

  // Payload support
  if b_PayloadSupport then

    // Use IF call as we are in RT
      s_PropertyValuePair.udPropertyId    := DO_PROP_READ_OFFSET;
      s_PropertyValuePair.udPropertyValue := udAddress;

      // us_ByteCnt: stays the same all the time

      MULTI_VARAN_iSetDoProperties(s_ISyncDO.p_Handle$UDINT, 1, #s_PropertyValuePair );

    s_ISyncDO.b_DOIsRunning.StartRequest := true;
  else
  //Set Address which should be read
  s_ISyncDO.p_DOSettings^.ud_Address := DeviceAddress + udAddress;

  //Set Length of Package
  s_ISyncDO.p_DOSettings^.us_ByteCnt := 2;

  //Start SingleRun of DataObject
  ResetDataObject(p_handleDO  := s_ISyncDO.p_Handle,
                  us_state    := VARAN_DO_SINGLE_RUN,
                  ud_bytes    := 2);
  end_if;

END_FUNCTION

FUNCTION VST011::CalcFrequencyLimits
VAR
  tmpCounter    : USINT;
  tmpFrequency  : UDINT;
END_VAR

  //Loop to check all FrequencyLimits
  //*****************************************************************************
  for tmpCounter := 0 to (sizeof(a_FrequencyLimit) / sizeof(a_FrequencyLimit[0])) - 1 do

    //Get the selected FrequencyLimit
    case tmpCounter of

      0:  tmpFrequency := FrequencyLimit1;
      1:  tmpFrequency := FrequencyLimit2;
      2:  tmpFrequency := FrequencyLimit4;
      3:  tmpFrequency := FrequencyLimit8;
      4:  tmpFrequency := FrequencyLimit16;
      5:  tmpFrequency := FrequencyLimit32;

    end_case;

    //Check if FrequencyLimit is active
    if tmpFrequency <> 16#FFFF_FFFF then

      //Calculate Hysterese
      //---------------------------------------------------------
      //LowLomit
      if tmpFrequency > FrequencyBandwidth / 2 then
        a_FrequencyLimit[tmpCounter].LimitLow := tmpFrequency - (FrequencyBandwidth / 2);
      else
        a_FrequencyLimit[tmpCounter].LimitLow := tmpFrequency;
      end_if;

      //High Limit
      if tmpFrequency + (FrequencyBandwidth / 2) < 1000000 then
        a_FrequencyLimit[tmpCounter].LimitHigh  := tmpFrequency + (FrequencyBandwidth / 2);
      else
        a_FrequencyLimit[tmpCounter].LimitHigh := tmpFrequency;
      end_if;

    else

      //Set Inactive
      a_FrequencyLimit[tmpCounter].LimitHigh  := 16#FFFF_FFFF;
      a_FrequencyLimit[tmpCounter].LimitLow   := 16#FFFF_FFFF;

    end_if;

  end_for;

  //*****************************************************************************

END_FUNCTION

FUNCTION GLOBAL VST011::SetStallCurrentWindow
  VAR_INPUT
    NewWindow   : UDINT;
  END_VAR

  udStallCurrentWindow := NewWindow;

END_FUNCTION

FUNCTION VIRTUAL GLOBAL VST011::Varan_HwInterrupt
  VAR_INPUT
    ud_reason   : UDINT;
    ud_data   : ^t_CallBackInterrupt;
  END_VAR
  VAR_OUTPUT
    sd_retval   : DINT;
  END_VAR

  SetDOsOff();
  sd_retval := Varan_Base::Varan_HwInterrupt(ud_reason:=ud_reason, ud_data:=ud_data);

END_FUNCTION

FUNCTION VIRTUAL GLOBAL VST011::GetDeviceID
  VAR_OUTPUT
    output  : UDINT;
  END_VAR

  output := VST011_DEVICE_ID;

END_FUNCTION

FUNCTION VIRTUAL GLOBAL VST011::CheckPostInitNeeded
	VAR_INPUT
		pbPostInitSettings 	: ^t_VM_CMD_NEED_POST_INIT_CALL_SETTINGS;
	END_VAR
	VAR_OUTPUT
		PostInitNeeded 	: BOOL;
	END_VAR

  if pbPostInitSettings <> NIL then
    pbPostInitSettings^ := 0;
  end_if;

  PostInitNeeded := TRUE;

END_FUNCTION
